# EPICS substitutions: iocBoot/iocvirPV/DPU02.substitutions
file "../../db/virAi.template"{ pattern
{DPU,	  num}
{02,	  0 }
{02,	  1 }
{02,	  2 }
{02,	  3 }
{02,	  4 }
{02,	  5 }
{02,	  6 }
{02,	  7 }
{02,	  8 }
{02,	  9 }
{02,	  10}
{02,	  11}
{02,	  12}
{02,	  13}
{02,	  14}
{02,	  15}
{02,	  16}
{02,	  17}
{02,	  18}
{02,	  19}
{02,	  20}
{02,	  21}
{02,	  22}
{02,	  23}
{02,	  24}
{02, 	  25}
{02,	  26}
{02,	  27}
{02,	  28}
{02,	  29}
{02,	  30}
{02,	  31}
{02,	  32}
{02,	  33}
{02,	  34}
{02,	  35}
{02,	  36}
{02,	  37}
{02,	  38}
{02,	  39}
{02,	  40}
{02,	  41}
{02,	  42}
{02,	  43}
{02,	  44}
{02,	  45}
{02,	  46}
{02,	  47}
{02,	  48}
{02,	  49}
{02,	  50}
{02,	  51}
{02,	  52}
{02,	  53}
{02,	  54}
{02,	  55}
{02,	  56}
{02,	  57}
{02,	  58}
{02,	  59}
{02,	  60}
{02,	  61}
{02,	  62}
{02, 	  63}
{02,      64}
{02,      65}
{02,      66}
{02,      67}
{02,      68}
{02,      69}
{02,      70}
{02,      71}
{02,      72}
{02,      73}
{02,      74}
{02,      75}
{02,      76}
{02,      77}
{02,      78}
{02,      79}
{02,      80}
{02,      81}
{02,      82}
{02,      83}
{02,      84}
{02,      85}
{02,      86}
{02,      87}
{02,      88}
{02,      89}
{02,      90}
{02,      91}
{02,      92}
{02,      93}
{02,      94}
{02,      95}
{02,      96}
{02,      97}
{02,      98}
{02,      99}
{02,     100}
{02,     101}
{02,     102}
{02,     103}
{02,     104}
{02,     105}
{02,     106}
{02,     107}
{02,     108}
{02,     109}
{02,     110}
{02,     111}
{02,     112}
{02,     113}
{02,     114}
{02,     115}
{02,     116}
{02,     117}
{02,     118}
{02,     119}
{02,     120}
{02,     121}
{02,     122}
{02,     123}
{02,     124}
{02,     125}
{02,     126}
{02,     127}
{02,     128}
{02,     129}
{02,     130}
{02,     131}
{02,     132}
{02,     133}
{02,     134}
{02,     135}
{02,     136}
{02,     137}
{02,     138}
{02,     139}
{02,     140}
{02,     141}
{02,     142}
{02,     143}
{02,     144}
{02,     145}
{02,     146}
{02,     147}
{02,     148}
{02,     149}
{02,     150}
{02,     151}
{02,     152}
{02,     153}
{02,     154}
{02,     155}
{02,     156}
{02,     157}
{02,     158}
{02,     159}
{02,     160}
{02,     161}
{02,     162}
{02,     163}
{02,     164}
{02,     165}
{02,     166}
{02,     167}
{02,     168}
{02,     169}
{02,     170}
{02,     171}
{02,     172}
{02,     173}
{02,     174}
{02,     175}
{02,     176}
{02,     177}
{02,     178}
{02,     179}
{02,     180}
{02,     181}
{02,     182}
{02,     183}
{02,     184}
{02,     185}
{02,     186}
{02,     187}
{02,     188}
{02,     189}
{02,     190}
{02,     191}
{02,     192}
{02,     193}
{02,     194}
{02,     195}
{02,     196}
{02,     197}
{02,     198}
{02,     199}
}
